# B&R Automation Studio project DriveControl
Automation Studio 4.2.5.388; Default project

## Configuration SampleText

CPU 4PP065.0571-P74, AutomationRuntime D4.52, Build 4.1.2, Vc V4.25.0, Safety 1.6

### Task classes (Cpu.sw)
```
Cyclic#1 (cycle 2000 us, tolerance 0 us):
  ncsdcctrl <- ncsdcctrl.prg
Cyclic#4:
  SDCAxisCtr <- SDCAxisCtrlX.prg
NcDataObjects: AcpParTab <- Libraries.AcpParTab.dob, acp10etxen <- acp10etxen.dob, gAxis01a <- gAxis01obj.gAxis01a.dob, gAxis01i <- gAxis01obj.gAxis01i.dob
Libraries: Acp10sdc, sys_lib, Runtime, asstring, Acp10man, Acp10par, NcGlobal, Acp10sim, Acp10_MC, brsystem, AsIOTime, AsBrStr, MotorContr
```

### Hardware
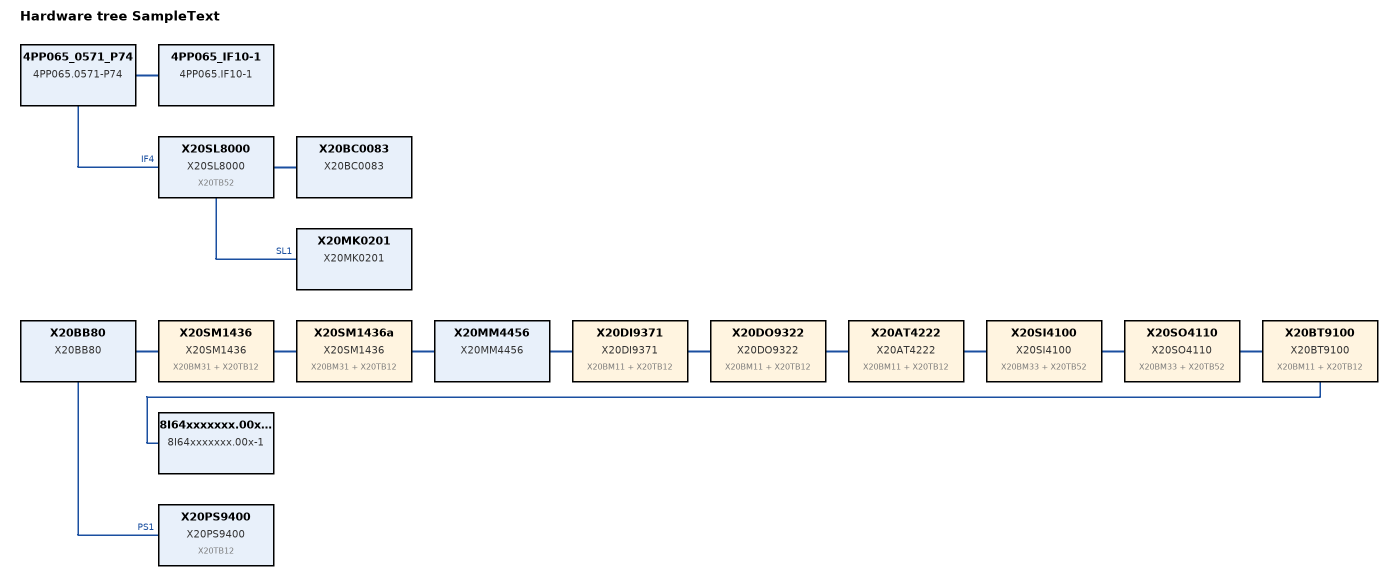
```
4PP065_0571_P74 : 4PP065.0571-P74 v1.1.2.0
  Connector IF4:
    EplInterfaceRedundant = 0
    EplEthInterfaceRedundant = 0
  Connector IF5:
    ActivateDevice = 1
    Mode = Manual
    InternetAddress = 10.1.1.13
    SubnetMask = 255.255.255.0
  ConfigurationID = DriveControl_SampleText
  Simulation = 1
  TimerDeviceType = EPLX2X
  TimerDevice = 4PP065_0571_P74.IF4
  TaskClassIdleTime = 2000
  Cyclic1Duration = 2000
  Cyclic1Tolerance = 0
  Cyclic1Output = 1
4PP065_IF10-1 : 4PP065.IF10-1 v1.0.3.0  [SS -> 4PP065_0571_P74.SS1]
8I64xxxxxxx.00x-1 : 8I64xxxxxxx.00x-1 v1.3.9.1  [X2X1 -> X20BT9100.X2X1 [Cable Type=X2XCable, Length=10, Version=1.0.0.2]]
  ActiveMotorSimulation_r1 = on
  BothEndSwitchesAreNormallyOpen_r1 = on
  QuickStopIsNormallyOpen_r1 = on
X20AT4222 : X20AT4222 v1.2.3.0  [SS1 -> X20TB12e.SS; SL -> X20BM11c.SL1]
X20BB80 : X20BB80 v1.0.2.0
X20BC0083 : X20BC0083 v2.7.0.0  [PLK1 -> X20SL8000.PLK2 (NodeNumber=2) [Cable Type=PowerlinkCable, Length=10, Version=1.0.0.2]; SL -> X20BB80.SL1]
X20BM11 : X20BM11 v1.0.0.1  [X2X1 -> X20BM33a.X2X2]
X20BM11a : X20BM11 v1.0.0.1  [X2X1 -> X20MM4456.X2X2]
X20BM11b : X20BM11 v1.0.0.1  [X2X1 -> X20BM11a.X2X2]
X20BM11c : X20BM11 v1.0.0.1  [X2X1 -> X20BM11b.X2X2]
X20BM31 : X20BM31 v1.0.0.1  [X2X1 -> X20BB80.IF1]
X20BM31a : X20BM31 v1.0.0.1  [X2X1 -> X20BM31.X2X2]
X20BM33 : X20BM33 v1.0.0.4  [X2X1 -> X20BM11c.X2X2]
X20BM33a : X20BM33 v1.0.0.4  [X2X1 -> X20BM33.X2X2]
X20BT9100 : X20BT9100 v1.0.3.0  [SS1 -> X20TB12f.SS; SL -> X20BM11.SL1]
X20DI9371 : X20DI9371 v1.0.2.0  [SS1 -> X20TB12c.SS; SL -> X20BM11a.SL1]
X20DO9322 : X20DO9322 v1.0.3.0  [SS1 -> X20TB12d.SS; SL -> X20BM11b.SL1]
X20MK0201 : X20MK0201 v1.0.0.0  [SL -> X20SL8000.SL1]
X20MM4456 : X20MM4456 v1.1.5.0  [X2X1 -> X20BM31a.X2X2]
X20PS9400 : X20PS9400 v1.0.2.4  [SS1 -> X20TB12.SS; PS -> X20BB80.PS1]
X20SI4100 : X20SI4100 v1.10.1.1  [SS1 -> X20TB52.SS; SL -> X20BM33.SL1]
X20SL8000 : X20SL8000 v1.6.5.1  [PLK1 -> 4PP065_0571_P74.IF4 (NodeNumber=1) [Cable Type=PowerlinkCable, Length=10, Version=1.0.0.2]; PLK2 -> X20BC0083.PLK1 (NodeNumber=1) [Cable Type=PowerlinkCable, Length=10, Version=1.0.0.2]; SS1 -> X20TB52b.SS]
  SafeProject = SafeLOGIC-1
X20SM1436 : X20SM1436 v1.4.2.1  [SS1 -> X20TB12a.SS; SL -> X20BM31.SL1]
X20SM1436a : X20SM1436 v1.4.2.1  [SS1 -> X20TB12b.SS; SL -> X20BM31a.SL1]
X20SO4110 : X20SO4110 v1.10.1.1  [SS1 -> X20TB52a.SS; SL -> X20BM33a.SL1]
  SafeModuleID = 3
X20TB12 : X20TB12 v1.0.0.0
X20TB12a : X20TB12 v1.0.0.0
X20TB12b : X20TB12 v1.0.0.0
X20TB12c : X20TB12 v1.0.0.0
X20TB12d : X20TB12 v1.0.0.0
X20TB12e : X20TB12 v1.0.0.0
X20TB12f : X20TB12 v1.0.0.0
X20TB52 : X20TB52 v1.0.0.1
X20TB52a : X20TB52 v1.0.0.1
X20TB52b : X20TB52 v1.0.0.1
```

### Acp10map.ncm - 4PP065_0571_P74/Motion/Acp10map.ncm
```
NcMapping (NcSwId=Acp10, DisabledNodesAreHidden=False)
  NcObject Axis_X (ModuleId=8I64xxxxxxx.00x-1, ModuleAddress=SDC_IF1.ST1, Type=ncAXIS, Channel=1, AcoposSimulation=Off, InitParameter=gAxis01i, AcoposParameter=gAxis01a, Disabled=FALSE, ModuleDisabled=FALSE)
```

## Configuration Simulation

CPU , AutomationRuntime J4.25

### Acp10map.ncm - PC_any/Acp10map.ncm
```
NcMapping (NcSwId=ACP10)
```

## Logical view

Binary libraries used (declarations not repeated): Runtime, Operator, AsIecCon, astime, sys_lib, asstring, Acp10man, Acp10par, NcGlobal, AsBrStr, Acp10sim, Acp10_MC, brsystem, Acp10sdc, AsIOTime

### Global.var - Global variables
```iecst
VAR
	gAxis01 : ACP10AXIS_typ := (0);
	gAxis01_HW : SdcHwCfg_typ := (0);
	gAxis01_DrvIf : SdcDrvIf16_typ := (0);
	gAxis01_DiDoIf : SdcDiDoIf_typ := (0);
	gAxis01_ModuleOk : BOOL := 0;
	gAxis_X_EncIf : SdcEncIf16_typ := (0);
END_VAR
```

### Package Logical/Libraries - Global libraries

### Data object Logical/Libraries/AcpParTab (Apt)

#### AcpParTab.apt - ACOPOS Parameter table
```
AcoposParameterTable:
  Root Parameters:
    64201 = 6500 (Name=SERVO_V_MAX_OUTPUT, Unit=Units/s)  // Servo drive adjustment: Velocity at maximum output value
    109 = 24 (Name=SCALE_ENCOD_INCR)  // Encoder1: Encoder scaling: increments per encoder revolution
```

### Library Logical/Libraries/MotorContr (ANSIC)

#### MotorContr.fun - Exported functions and function blocks
```iecst
FUNCTION_BLOCK FB_Regulator (*Regulator functional block*) (*$GROUP=User,$CAT=User,$GROUPICON=User.png,$CATICON=User.png*)
	VAR_INPUT
		e : REAL; (*Mismatch between the reference action and the real speed of rotation of the DCM shaft [rpm]*)
	END_VAR
	VAR_OUTPUT
		u : REAL; (*Voltage supplied to the DCM input [V]*)
	END_VAR
	VAR
		k_p : REAL; (*Regulator proportional gain*)
		k_i : REAL; (*Integral gain of the regulator*)
		integrator : FB_Integrator; (*Integrator*)
		iyOld : REAL; (*Storing the previous value of the anti-accumulation scheme*)
		max_abs_value : REAL; (*Limit block boundary [B]*)
		dt : REAL; (*Calculation step [s]*)
		e_p : REAL; (*Temporary variable [rpm]*)
	END_VAR
END_FUNCTION_BLOCK

FUNCTION_BLOCK FB_Motor (*Motor functional block*) (*$GROUP=User,$CAT=User,$GROUPICON=User.png,$CATICON=User.png*)
	VAR_INPUT
		u : REAL; (*Input voltage [V]*)
	END_VAR
	VAR_OUTPUT
		w : REAL; (*Rotation frequency [rpm]*)
		phi : REAL; (*Position [rad]*)
	END_VAR
	VAR
		integrator : FB_Integrator; (*Integrator*)
		Tm : REAL; (*Electromechanical time constant [s]*)
		ke : REAL; (*Constant EMF of the motor [V * min/rev]*)
		dt : REAL; (*Calculation step [s]*)
	END_VAR
END_FUNCTION_BLOCK

FUNCTION_BLOCK FB_Integrator (*Integrator functional block*) (*$GROUP=User,$CAT=User,$GROUPICON=User.png,$CATICON=User.png*)
	VAR_INPUT
		in : REAL; (*Integrator input*)
	END_VAR
	VAR_OUTPUT
		out : REAL; (*Integrator output*)
	END_VAR
	VAR
		dt : REAL; (*Calculation step [s]*)
	END_VAR
END_FUNCTION_BLOCK

{REDUND_ERROR} FUNCTION_BLOCK FB_Axis (* *) (*$GROUP=User,$CAT=User,$GROUPICON=User.png,$CATICON=User.png*)
	VAR_INPUT
		reset_error : {REDUND_UNREPLICABLE} BOOL;
		endswitch_a_reached : {REDUND_UNREPLICABLE} BOOL;
		endswitch_b_reached : {REDUND_UNREPLICABLE} BOOL;
	END_VAR
	VAR_OUTPUT
		reset_counter : {REDUND_UNREPLICABLE} BOOL;
		pwm_value : {REDUND_UNREPLICABLE} INT;
		counter : {REDUND_UNREPLICABLE} INT;
		speed : {REDUND_UNREPLICABLE} REAL;
	END_VAR
	VAR
		last_counter : {REDUND_UNREPLICABLE} INT;
		desired_speed : {REDUND_UNREPLICABLE} REAL;
		regulator : {REDUND_UNREPLICABLE} FB_Regulator;
		dt : REAL;
	END_VAR
	VAR_INPUT
		u : REAL;
	END_VAR
END_FUNCTION_BLOCK
```

#### FB_Motor.c
```c
#include <bur/plctypes.h>
#ifdef __cplusplus
	extern "C"
	{
#endif
	#include "MotorContr.h"
#ifdef __cplusplus
	};
#endif
/* This function is a model of the control object (DC motor) */
void FB_Motor(struct FB_Motor* inst)
{
	inst->integrator.in = (inst->u*(1/inst->ke) - inst->w)*(inst->dt/inst->Tm);
	FB_Integrator(&(inst->integrator));
	inst->w = inst->integrator.out;

	inst->integrator.in = inst->w*inst->dt;
	FB_Integrator(&(inst->integrator));
	inst->phi = inst->integrator.out;
}
```

#### FB_Regulator.c
```c
#include <bur/plctypes.h>
#ifdef __cplusplus
	extern "C"
	{
#endif
	#include "MotorContr.h"
#ifdef __cplusplus
	};
#endif
/* This function is a PI controller model */
void FB_Regulator(struct FB_Regulator* inst)
{
	inst->integrator.in = inst->e*inst->k_i*inst->dt + inst->iyOld;
	FB_Integrator(&(inst->integrator));

	inst->e_p = inst->e*inst->k_p;

	if(inst->e_p < inst->max_abs_value || inst->e_p > -inst->max_abs_value);
	else
	{
		if(inst->e_p > 0) inst->e_p = inst->max_abs_value;
		else inst->e_p = -inst->max_abs_value;
	}

	inst->e_p += inst->integrator.out;

	if(inst->e_p < inst->max_abs_value || inst->e_p > -inst->max_abs_value)
		inst->u = inst->e_p;
	else
	{
		if(inst->e_p > 0) inst->u = inst->max_abs_value;
		else inst->u = -inst->max_abs_value;
	}

	inst->iyOld = inst->u - inst->e_p;
}
```

#### FB_Integrator.c
```c
#include <bur/plctypes.h>
#ifdef __cplusplus
	extern "C"
	{
#endif
	#include "MotorContr.h"
#ifdef __cplusplus
	};
#endif
/* This function is an integrator */
void FB_Integrator(struct FB_Integrator* inst)
{
	inst->out += inst->in;
}
```

#### FB_Axis.c
```c
#include <bur/plctypes.h>
#ifdef __cplusplus
	extern "C"
	{
#endif
	#include "MotorContr.h"
#ifdef __cplusplus
	};
#endif
void FB_Axis(struct FB_Axis* inst)
{
	inst->pwm_value = (inst->u/24)*32767;
	inst->speed = ((REAL)inst->counter - (REAL)inst->last_counter)*3000/(24.0*inst->dt); //counter - last_counter
	inst->last_counter=inst->counter;
}
```

### Package Logical/gAxis01obj - gAxis01obj

### gAxis01a.apt
```
AcoposParameterTable:
  Root Parameters:
    230 = PCTRL_S_SET (Name=PCTRL_S_ACT_PARID)
    110 = ncSW_ON (Name=CMD_SIMULATION)
    64201 = 546116.666666667 (Name=SERVO_V_MAX_OUTPUT)
```

### gAxis01i.ax
```
InitParameter (Version=5.02.1, NcSwId=Acp10)
  ACP10AXIS_typ:
    dig_in:
      level:
        reference = ncACTIV_HI
        pos_hw_end = ncACTIV_HI
        neg_hw_end = ncACTIV_HI
        trigger1 = ncACTIV_HI
        trigger2 = ncACTIV_HI
    encoder_if:
      parameter:
        count_dir = ncSTANDARD
        scaling:
          load:
            units = 3000
            rev_motor = 1
    limit:
      parameter:
        v_pos = 10000
        v_neg = 10000
        a1_pos = 10000.0
        a2_pos = 10000.0
        a1_neg = 10000.0
        a2_neg = 10000.0
        t_jolt = 0
        t_in_pos = 0
        pos_sw_end = 2000000000
        neg_sw_end = -2000000000
        ds_warning = 500
        ds_stop = 50000.0
        a_stop = 1.0e30
        dv_stop = 0
        dv_stop_mode = ncOFF
    controller:
      mode = ncPOSITION + ncFF
      position:
        kv = 10.0
        tn = 0
        t_predict = 0.01
        t_total = 0.01
        p_max = 1.0e30
        i_max = 0
      speed:
        kv = 10.0
        tn = 0
        t_filter = 0.0
        isq_filter1:
          type = ncOFF
          a0 = 0.0
          a1 = 0.0
          b0 = 0.0
          b1 = 0.0
          b2 = 0.0
          c0_par_id = 0
          c1_par_id = 0
        isq_filter2:
          type = ncOFF
          a0 = 0.0
          a1 = 0.0
          b0 = 0.0
          b1 = 0.0
          b2 = 0.0
          c0_par_id = 0
          c1_par_id = 0
        isq_filter3:
          type = ncOFF
          a0 = 0.0
          a1 = 0.0
          b0 = 0.0
          b1 = 0.0
          b2 = 0.0
          c0_par_id = 0
          c1_par_id = 0
      uf:
        type = ncLINEAR + ncCORRECTION
        auto_config = ncMOTOR_PAR
        u0 = 0
        un = 0
        fn = 50.0
        k_f_slip = 0
      ff:
        torque_load = 0.0
        torque_pos = 0.0
        torque_neg = 0.0
        kv_torque = 0.0
        inertia = 0.0
        t_filter_a = 0.0
    move:
      stop:
        parameter[0]:
          decel_ramp = ncA_LIMIT
          controller = ncON
        parameter[1]:
          decel_ramp = ncA_LIMIT
          controller = ncON
        parameter[2]:
          decel_ramp = ncA_LIMIT
          controller = ncON
        parameter[3]:
          decel_ramp = ncA_LIMIT
          controller = ncON
        quickstop:
          decel_ramp = ncA_LIMIT
          t_jolt = 0
        drive_error:
          decel_ramp = ncA_LIMIT
      homing:
        parameter:
          s = 0
          v_switch = 6000.0
          v_trigger = 2000.0
          a = 10000.0
          mode = ncEND_SWITCH
          edge_sw = ncNEGATIVE
          start_dir = ncPOSITIVE
          trigg_dir = ncNEGATIVE
          ref_pulse = ncOFF
          fix_dir = ncOFF
          tr_s_block = 0
          torque_lim = 0
          ds_block = 0
          ds_stop = 0
      basis:
        parameter:
          v_pos = 5000
          v_neg = 5000
          a1_pos = 10000.0
          a2_pos = 10000.0
          a1_neg = 10000.0
          a2_neg = 10000.0
    message:
      text:
        parameter:
          format = ncBREAK
          columns = 80
          data_modul = acp10etxen
```

### Program Logical/SDCAxisCtrlX (ANSIC)

#### Variables.var
```iecst
VAR
	temp : REAL := 0.0;
	axis_X : FB_Axis := (0);
	coil_powered : BOOL := FALSE;
	coil_pwm_value : INT := 0;
	fb_controller : FB_Regulator := (0);
END_VAR
```

#### Main.c
```c
#include <bur/plctypes.h>

#ifdef _DEFAULT_INCLUDES
	#include <AsDefault.h>
#endif

void _INIT ProgramInit(void)
{
	gAxis01_HW.EncIf1_Typ = ncSDC_ENC16;
	gAxis01_HW.DiDoIf_Typ = ncSDC_DIDO;
	gAxis01_HW.DrvIf_Typ = ncSDC_DRVSERVO16;

	gAxis_X_EncIf.iEncOK = 1;
	gAxis01_DrvIf.iDrvOK = 1;
	gAxis01_DrvIf.iStatusEnable = 1;
	gAxis01_DiDoIf.iDriveReady = 1;
	fb_controller.dt = 0.002;
	fb_controller.k_i = 0.16;
	fb_controller.k_p = 0.0064;
	fb_controller.max_abs_value = 24.0;
//	pwm_period = 200;
}

void _CYCLIC ProgramCyclic(void)
{
	if (!coil_powered) coil_pwm_value = 0;
	else coil_pwm_value = 32767;
	gAxis_X_EncIf.iLifeCnt++;
	gAxis01_DiDoIf.iLifeCntDriveEnable++;
	gAxis01_DiDoIf.iLifeCntDriveReady++;
	gAxis01_DiDoIf.iLifeCntNegHwEnd++;
	gAxis01_DiDoIf.iLifeCntPosHwEnd++;
	gAxis01_DiDoIf.iLifeCntReference++;
	gAxis01_DrvIf.iLifeCnt++;
	gAxis_X_EncIf.iActTime = (INT)AsIOTimeCyclicStart();
	gAxis_X_EncIf.iActPos = axis_X.counter;
	temp = gAxis01_DrvIf.oSetPos;
	fb_controller.e = (temp/32767.0)*6500.0 - axis_X.speed;
	FB_Regulator(&fb_controller);
	axis_X.u = fb_controller.u;
	gAxis01_DiDoIf.iPosHwEnd = axis_X.endswitch_b_reached;
	gAxis01_DiDoIf.iNegHwEnd = axis_X.endswitch_a_reached;
	if(axis_X.endswitch_a_reached) axis_X.reset_error = 1;
	if(axis_X.endswitch_b_reached) axis_X.reset_error = 1;
	axis_X.reset_error = 0;
}

void _EXIT ProgramExit(void)
{

}
```

Listed in the project but not available here: Logical/Global.typ, Logical/Libraries/MotorContr/Types.typ, Logical/Libraries/MotorContr/Constants.var, Logical/ncsdcctrl, Logical/acp10etxen
